(* CODESYS project Avangard(contr1).project
   Title: Avangard(contr1)
   Version: 0.0.0.0
   Author: Administrator

Project tree, tasks and I/O mapping:
  MyController : TM241CE40T/U, Schneider Electric, order no. TM241CE40T/U, version 4.0.6.18
    application Application
      task MAST (cyclic, interval 20 ms, priority 15, watchdog 100 ms x 1) calls MainPrgY, MainLD, MainPrgX
      global variables GVL
    DI : Digital Inputs, Schneider Electric, version 4.0.6.18
        input  idwDI_IDW0 : DWORD  // IDW0
        input  Application.X01_0 : BOOL  // IDW0.I0
        input  Application.X01_1 : BOOL  // IDW0.I1
        input  Application.X01_2 : BOOL  // IDW0.I2
        input  Application.X01_3 : BOOL  // IDW0.I3
        input  Application.X01_4 : BOOL  // IDW0.I4
        input  Application.X01_5 : BOOL  // IDW0.I5
        input  Application.X01_6 : BOOL  // IDW0.I6
        input  Application.X01_7 : BOOL  // IDW0.I7
        input  Application.X01_8 : BOOL  // IDW0.I8
        input  Application.X01_9 : BOOL  // IDW0.I9
        input  Application.X01_10 : BOOL  // IDW0.I10
        input  Application.X01_11 : BOOL  // IDW0.I11
        input  Application.X01_12 : BOOL  // IDW0.I12
        input  Application.X01_13 : BOOL  // IDW0.I13
        input  Application.X01_14 : BOOL  // IDW0.I14
        input  Application.X01_15 : BOOL  // IDW0.I15
        input  Application.X01_16 : BOOL  // IDW0.I16
        input  Application.X01_17 : BOOL  // IDW0.I17
        input  Application.X01_18 : BOOL  // IDW0.I18
        input  Application.X01_19 : BOOL  // IDW0.I19
        input  Application.X01_20 : BOOL  // IDW0.I20
        input  Application.X01_21 : BOOL  // IDW0.I21
        input  Application.X01_22 : BOOL  // IDW0.I22
        input  Application.X01_23 : BOOL  // IDW0.I23
        input  ibDI_IB1 : BYTE  // IB1
    DQ : Digital Outputs, Schneider Electric, version 4.0.6.18
        output Application.Y01_0 : BOOL  // QW0.Q0
        output Application.Y01_1 : BOOL  // QW0.Q1
        output Application.Y01_2 : BOOL  // QW0.Q2
        output Application.Y01_3 : BOOL  // QW0.Q3
        output Application.Y01_4 : BOOL  // QW0.Q4
        output Application.Y01_5 : BOOL  // QW0.Q5
        output Application.Y01_6 : BOOL  // QW0.Q6
        output Application.Y01_7 : BOOL  // QW0.Q7
        output Application.Y01_8 : BOOL  // QW0.Q8
        output Application.Y01_9 : BOOL  // QW0.Q9
        output Application.Y01_10 : BOOL  // QW0.Q10
        output Application.Y01_11 : BOOL  // QW0.Q11
        output Application.Y01_12 : BOOL  // QW0.Q12
        output Application.Y01_13 : BOOL  // QW0.Q13
        output Application.Y01_14 : BOOL  // QW0.Q14
        output Application.Y01_15 : BOOL  // QW0.Q15
        output qbDQ_QB1 : BYTE  // QB1
        unmapped channels: QW0
    Counters : Counters, Schneider Electric, version 4.0.6.18
    Pulse_Generators : Pulse Generators, Schneider Electric, version 4.0.6.18
    Cartridge_1 : Cartridge, Schneider Electric, version 4.0.6.18
    Cartridge_2 : Cartridge, Schneider Electric, version 4.0.6.18
    IO_Bus : IO bus - TM3, Schneider Electric, version 4.0.6.18
      Module_1 : TM3DI32K, Schneider Electric, order no. TM3DI32K, version 1.0.1.3
          input  idwModule_1_ID0 : DWORD  // ID0
          input  Application.X11_0 : BOOL  // ID0.I0
          input  Application.X11_1 : BOOL  // ID0.I1
          input  Application.X11_2 : BOOL  // ID0.I2
          input  Application.X11_3 : BOOL  // ID0.I3
          input  Application.X11_4 : BOOL  // ID0.I4
          input  Application.X11_5 : BOOL  // ID0.I5
          input  Application.X11_6 : BOOL  // ID0.I6
          input  Application.X11_7 : BOOL  // ID0.I7
          input  Application.X11_8 : BOOL  // ID0.I8
          input  Application.X11_9 : BOOL  // ID0.I9
          input  Application.X11_10 : BOOL  // ID0.I10
          input  Application.X11_11 : BOOL  // ID0.I11
          input  Application.X11_12 : BOOL  // ID0.I12
          input  Application.X11_13 : BOOL  // ID0.I13
          input  Application.X11_14 : BOOL  // ID0.I14
          input  Application.X11_15 : BOOL  // ID0.I15
          input  Application.X11_16 : BOOL  // ID0.I16
          input  Application.X11_17 : BOOL  // ID0.I17
          input  Application.X11_18 : BOOL  // ID0.I18
          input  Application.X11_19 : BOOL  // ID0.I19
          input  Application.X11_20 : BOOL  // ID0.I20
          input  Application.X11_21 : BOOL  // ID0.I21
          input  Application.X11_22 : BOOL  // ID0.I22
          input  Application.X11_23 : BOOL  // ID0.I23
          input  Application.X11_24 : BOOL  // ID0.I24
          input  Application.X11_25 : BOOL  // ID0.I25
          input  Application.X11_26 : BOOL  // ID0.I26
          input  Application.X11_27 : BOOL  // ID0.I27
          input  Application.X11_28 : BOOL  // ID0.I28
          input  Application.X11_29 : BOOL  // ID0.I29
          input  Application.X11_30 : BOOL  // ID0.I30
          input  Application.X11_31 : BOOL  // ID0.I31
      Module_2 : TM3DI32K, Schneider Electric, order no. TM3DI32K, version 1.0.1.3
          input  Application.X12_0 : BOOL  // ID0.I0
          input  Application.X12_1 : BOOL  // ID0.I1
          input  Application.X12_2 : BOOL  // ID0.I2
          input  Application.X12_3 : BOOL  // ID0.I3
          input  Application.X12_4 : BOOL  // ID0.I4
          input  Application.X12_5 : BOOL  // ID0.I5
          input  Application.X12_6 : BOOL  // ID0.I6
          input  Application.X12_7 : BOOL  // ID0.I7
          input  Application.X12_8 : BOOL  // ID0.I8
          input  Application.X12_9 : BOOL  // ID0.I9
          input  Application.X12_10 : BOOL  // ID0.I10
          input  Application.X12_11 : BOOL  // ID0.I11
          input  Application.X12_12 : BOOL  // ID0.I12
          input  Application.X12_13 : BOOL  // ID0.I13
          input  Application.X12_14 : BOOL  // ID0.I14
          input  Application.X12_15 : BOOL  // ID0.I15
          input  Application.X12_16 : BOOL  // ID0.I16
          input  Application.X12_17 : BOOL  // ID0.I17
          input  Application.X12_18 : BOOL  // ID0.I18
          input  Application.X12_19 : BOOL  // ID0.I19
          input  Application.X12_20 : BOOL  // ID0.I20
          input  Application.X12_21 : BOOL  // ID0.I21
          input  Application.X12_22 : BOOL  // ID0.I22
          input  Application.X12_23 : BOOL  // ID0.I23
          input  Application.X12_24 : BOOL  // ID0.I24
          input  Application.X12_25 : BOOL  // ID0.I25
          input  Application.X12_26 : BOOL  // ID0.I26
          input  Application.X12_27 : BOOL  // ID0.I27
          input  Application.X12_28 : BOOL  // ID0.I28
          input  Application.X12_29 : BOOL  // ID0.I29
          input  Application.X12_30 : BOOL  // ID0.I30
          input  Application.X12_31 : BOOL  // ID0.I31
          unmapped channels: ID0
      Module_5 : TM3DI32K, Schneider Electric, order no. TM3DI32K, version 1.0.1.3
          input  Application.X15_0 : BOOL  // ID0.I0
          input  Application.X15_1 : BOOL  // ID0.I1
          input  Application.X15_2 : BOOL  // ID0.I2
          input  Application.X15_3 : BOOL  // ID0.I3
          input  Application.X15_4 : BOOL  // ID0.I4
          input  Application.X15_5 : BOOL  // ID0.I5
          input  Application.X15_6 : BOOL  // ID0.I6
          input  Application.X15_7 : BOOL  // ID0.I7
          input  Application.X15_8 : BOOL  // ID0.I8
          input  Application.X15_9 : BOOL  // ID0.I9
          input  Application.X15_10 : BOOL  // ID0.I10
          input  Application.X15_11 : BOOL  // ID0.I11
          input  Application.X15_12 : BOOL  // ID0.I12
          input  Application.X15_13 : BOOL  // ID0.I13
          input  Application.X15_14 : BOOL  // ID0.I14
          input  Application.X15_15 : BOOL  // ID0.I15
          input  Application.X15_16 : BOOL  // ID0.I16
          input  Application.X15_17 : BOOL  // ID0.I17
          input  Application.X15_18 : BOOL  // ID0.I18
          input  Application.X15_19 : BOOL  // ID0.I19
          input  Application.X15_20 : BOOL  // ID0.I20
          input  Application.X15_21 : BOOL  // ID0.I21
          input  Application.X15_22 : BOOL  // ID0.I22
          input  Application.X15_23 : BOOL  // ID0.I23
          input  Application.X15_24 : BOOL  // ID0.I24
          input  Application.X15_25 : BOOL  // ID0.I25
          input  Application.X15_26 : BOOL  // ID0.I26
          input  Application.X15_27 : BOOL  // ID0.I27
          input  Application.X15_28 : BOOL  // ID0.I28
          input  Application.X15_29 : BOOL  // ID0.I29
          input  Application.X15_30 : BOOL  // ID0.I30
          input  Application.X15_31 : BOOL  // ID0.I31
          unmapped channels: ID0
      Module_4 : TM3DI32K, Schneider Electric, order no. TM3DI32K, version 1.0.1.3
          input  Application.X14_0 : BOOL  // ID0.I0
          input  Application.X14_1 : BOOL  // ID0.I1
          input  Application.X14_2 : BOOL  // ID0.I2
          input  Application.X14_3 : BOOL  // ID0.I3
          input  Application.X14_4 : BOOL  // ID0.I4
          input  Application.X14_5 : BOOL  // ID0.I5
          input  Application.X14_6 : BOOL  // ID0.I6
          input  Application.X14_7 : BOOL  // ID0.I7
          input  Application.X14_8 : BOOL  // ID0.I8
          input  Application.X14_9 : BOOL  // ID0.I9
          input  Application.X14_10 : BOOL  // ID0.I10
          input  Application.X14_11 : BOOL  // ID0.I11
          input  Application.X14_12 : BOOL  // ID0.I12
          input  Application.X14_13 : BOOL  // ID0.I13
          input  Application.X14_14 : BOOL  // ID0.I14
          input  Application.X14_15 : BOOL  // ID0.I15
          input  Application.X14_16 : BOOL  // ID0.I16
          input  Application.X14_17 : BOOL  // ID0.I17
          input  Application.X14_18 : BOOL  // ID0.I18
          input  Application.X14_19 : BOOL  // ID0.I19
          input  Application.X14_20 : BOOL  // ID0.I20
          input  Application.X14_21 : BOOL  // ID0.I21
          input  Application.X14_22 : BOOL  // ID0.I22
          input  Application.X14_23 : BOOL  // ID0.I23
          input  Application.X14_24 : BOOL  // ID0.I24
          input  Application.X14_25 : BOOL  // ID0.I25
          input  Application.X14_26 : BOOL  // ID0.I26
          input  Application.X14_27 : BOOL  // ID0.I27
          input  Application.X14_28 : BOOL  // ID0.I28
          input  Application.X14_29 : BOOL  // ID0.I29
          input  Application.X14_30 : BOOL  // ID0.I30
          input  Application.X14_31 : BOOL  // ID0.I31
          unmapped channels: ID0
      Module_3 : TM3DI32K, Schneider Electric, order no. TM3DI32K, version 1.0.1.3
          input  Application.X13_0 : BOOL  // ID0.I0
          input  Application.X13_1 : BOOL  // ID0.I1
          input  Application.X13_2 : BOOL  // ID0.I2
          input  Application.X13_3 : BOOL  // ID0.I3
          input  Application.X13_4 : BOOL  // ID0.I4
          input  Application.X13_5 : BOOL  // ID0.I5
          input  Application.X13_6 : BOOL  // ID0.I6
          input  Application.X13_7 : BOOL  // ID0.I7
          input  Application.X13_8 : BOOL  // ID0.I8
          input  Application.X13_9 : BOOL  // ID0.I9
          input  Application.X13_10 : BOOL  // ID0.I10
          input  Application.X13_11 : BOOL  // ID0.I11
          input  Application.X13_12 : BOOL  // ID0.I12
          input  Application.X13_13 : BOOL  // ID0.I13
          input  Application.X13_14 : BOOL  // ID0.I14
          input  Application.X13_15 : BOOL  // ID0.I15
          input  Application.X13_16 : BOOL  // ID0.I16
          input  Application.X13_17 : BOOL  // ID0.I17
          input  Application.X13_18 : BOOL  // ID0.I18
          input  Application.X13_19 : BOOL  // ID0.I19
          input  Application.X13_20 : BOOL  // ID0.I20
          input  Application.X13_21 : BOOL  // ID0.I21
          input  Application.X13_22 : BOOL  // ID0.I22
          input  Application.X13_23 : BOOL  // ID0.I23
          input  Application.X13_24 : BOOL  // ID0.I24
          input  Application.X13_25 : BOOL  // ID0.I25
          input  Application.X13_26 : BOOL  // ID0.I26
          input  Application.X13_27 : BOOL  // ID0.I27
          input  Application.X13_28 : BOOL  // ID0.I28
          input  Application.X13_29 : BOOL  // ID0.I29
          input  Application.X13_30 : BOOL  // ID0.I30
          input  Application.X13_31 : BOOL  // ID0.I31
          unmapped channels: ID0
      Module_6 : TM3DQ32TK, Schneider Electric, order no. TM3DQ32TK, version 1.0.1.3
          output Application.Y16_0 : BOOL  // QD0.Q0
          output Application.Y16_1 : BOOL  // QD0.Q1
          output Application.Y16_2 : BOOL  // QD0.Q2
          output Application.Y16_3 : BOOL  // QD0.Q3
          output Application.Y16_4 : BOOL  // QD0.Q4
          output Application.Y16_5 : BOOL  // QD0.Q5
          output Application.Y16_6 : BOOL  // QD0.Q6
          output Application.Y16_7 : BOOL  // QD0.Q7
          output Application.Y16_8 : BOOL  // QD0.Q8
          output Application.Y16_9 : BOOL  // QD0.Q9
          output Application.Y16_10 : BOOL  // QD0.Q10
          output Application.Y16_11 : BOOL  // QD0.Q11
          output Application.Y16_12 : BOOL  // QD0.Q12
          output Application.Y16_13 : BOOL  // QD0.Q13
          output Application.Y16_14 : BOOL  // QD0.Q14
          output Application.Y16_15 : BOOL  // QD0.Q15
          output Application.Y16_16 : BOOL  // QD0.Q16
          output Application.Y16_17 : BOOL  // QD0.Q17
          output Application.Y16_18 : BOOL  // QD0.Q18
          output Application.Y16_19 : BOOL  // QD0.Q19
          output Application.Y16_20 : BOOL  // QD0.Q20
          output Application.Y16_21 : BOOL  // QD0.Q21
          output Application.Y16_22 : BOOL  // QD0.Q22
          output Application.Y16_23 : BOOL  // QD0.Q23
          output Application.Y16_24 : BOOL  // QD0.Q24
          output Application.Y16_25 : BOOL  // QD0.Q25
          output Application.Y16_26 : BOOL  // QD0.Q26
          output Application.Y16_27 : BOOL  // QD0.Q27
          output Application.Y16_28 : BOOL  // QD0.Q28
          output Application.Y16_29 : BOOL  // QD0.Q29
          output Application.Y16_30 : BOOL  // QD0.Q30
          output Application.Y16_31 : BOOL  // QD0.Q31
          unmapped channels: QD0
      Module_7 : TM3DQ32TK, Schneider Electric, order no. TM3DQ32TK, version 1.0.1.3
          output Application.Y17_0 : BOOL  // QD0.Q0
          output Application.Y17_1 : BOOL  // QD0.Q1
          output Application.Y17_2 : BOOL  // QD0.Q2
          output Application.Y17_3 : BOOL  // QD0.Q3
          output Application.Y17_4 : BOOL  // QD0.Q4
          output Application.Y17_5 : BOOL  // QD0.Q5
          output Application.Y17_6 : BOOL  // QD0.Q6
          output Application.Y17_7 : BOOL  // QD0.Q7
          output Application.Y17_8 : BOOL  // QD0.Q8
          output Application.Y17_9 : BOOL  // QD0.Q9
          output Application.Y17_10 : BOOL  // QD0.Q10
          output Application.Y17_11 : BOOL  // QD0.Q11
          output Application.Y17_12 : BOOL  // QD0.Q12
          output Application.Y17_13 : BOOL  // QD0.Q13
          output Application.Y17_14 : BOOL  // QD0.Q14
          output Application.Y17_15 : BOOL  // QD0.Q15
          output Application.Y17_16 : BOOL  // QD0.Q16
          output Application.Y17_17 : BOOL  // QD0.Q17
          output Application.Y17_18 : BOOL  // QD0.Q18
          output Application.Y17_19 : BOOL  // QD0.Q19
          output Application.Y17_20 : BOOL  // QD0.Q20
          output Application.Y17_21 : BOOL  // QD0.Q21
          output Application.Y17_22 : BOOL  // QD0.Q22
          output Application.Y17_23 : BOOL  // QD0.Q23
          output Application.Y17_24 : BOOL  // QD0.Q24
          output Application.Y17_25 : BOOL  // QD0.Q25
          output Application.Y17_26 : BOOL  // QD0.Q26
          output Application.Y17_27 : BOOL  // QD0.Q27
          output Application.Y17_28 : BOOL  // QD0.Q28
          output Application.Y17_29 : BOOL  // QD0.Q29
          output Application.Y17_30 : BOOL  // QD0.Q30
          output Application.Y17_31 : BOOL  // QD0.Q31
          unmapped channels: QD0
    COM_Bus : COM bus, Schneider Electric, version 4.0.6.18
    Ethernet_1 : Ethernet Network, Schneider Electric, version 4.0.6.18
        settings: IPAddress = [192, 168, 1, 201]; SubnetMask = [255, 255, 255, 0]; GatewayAddress = [192, 168, 1, 1]; DeviceName = 'TM241CE40T_1'; WebServer = FALSE; FTP Server = FALSE; SoMachine Protocol = TRUE; Modbus Server = TRUE; NetManage Protocol = TRUE; SNMP protocol = FALSE; Enable Routing = FALSE; WebVisu protocol = FALSE; DHCP Server Active = FALSE
    Serial_Line_1 : Serial line, Schneider Electric, version 4.0.6.18
      SoMachine_Network_Manager : SoMachine-Network Manager, Schneider Electric, version 4.0.0.2
    Serial_Line_2 : Serial line, Schneider Electric, version 4.0.6.18
      Modbus_Manager : Modbus Manager, Schneider Electric, version 4.0.0.2
  libraries: Standard, * (System)
  program MainPrgY [ST]
  program MainLD [LD]
  function block DKS [LD]
  program MainPrgX [ST]
*)

// MyController/Application/GVL
VAR_GLOBAL
	XX AT %MW0 : ARRAY[0..11] OF WORD;  //данные с 1го контроллера
	YY AT %MW12 : ARRAY[0..5] OF WORD;  //данные для 1го контроллера на управление

	DKS_Time : WORD := 3;	//время срабатывания ДКС в сек
	
	Nor10200_DKS : BOOL;
	Nor10400_DKS : BOOL;
	Tr10500_DKS : BOOL;
	Tr10600_DKS : BOOL;
	Tr10700_DKS : BOOL;
	Tr20110_DKS : BOOL;
	Nor20300_DKS : BOOL;
	Nor21200_DKS : BOOL;
	Tr21300_DKS : BOOL;
	Tr30400_DKS : BOOL;
	Nor30500_DKS : BOOL;
	Tr30340_DKS : BOOL;
	Tr30700_DKS : BOOL;
	Nor40100_DKS : BOOL;
	
	
	// Контроллер 1
		//Входа
			X01_0 : BOOL;
			X01_1 : BOOL;
			X01_2 : BOOL;
			X01_3 : BOOL;
			X01_4 : BOOL;
			X01_5 : BOOL;
			X01_6 : BOOL;
			X01_7 : BOOL;
			X01_8 : BOOL;
			X01_9 : BOOL;
			X01_10 : BOOL;
			X01_11 : BOOL;
			X01_12 : BOOL;
			X01_13 : BOOL;
			X01_14 : BOOL;
			X01_15 : BOOL;
			X01_16 : BOOL;
			X01_17 : BOOL;
			X01_18 : BOOL;
			X01_19 : BOOL;
			X01_20 : BOOL;
			X01_21 : BOOL;
			X01_22 : BOOL;
			X01_23 : BOOL;
			X01_24 : BOOL;
			X01_25 : BOOL;
			X01_26 : BOOL;
			X01_27 : BOOL;
			X01_28 : BOOL;
			X01_29 : BOOL;
			X01_30 : BOOL;
			X01_31 : BOOL;
		//Выхода
			Y01_0 : BOOL;
			Y01_1 : BOOL;
			Y01_2 : BOOL;
			Y01_3 : BOOL;
			Y01_4 : BOOL;
			Y01_5 : BOOL;
			Y01_6 : BOOL;
			Y01_7 : BOOL;
			Y01_8 : BOOL;
			Y01_9 : BOOL;
			Y01_10 : BOOL;
			Y01_11 : BOOL;
			Y01_12 : BOOL;
			Y01_13 : BOOL;
			Y01_14 : BOOL;
			Y01_15 : BOOL;
			Y01_16 : BOOL;
			Y01_17 : BOOL;
			Y01_18 : BOOL;
			Y01_19 : BOOL;
			Y01_20 : BOOL;
			Y01_21 : BOOL;
			Y01_22 : BOOL;
			Y01_23 : BOOL;
			Y01_24 : BOOL;
			Y01_25 : BOOL;
			Y01_26 : BOOL;
			Y01_27 : BOOL;
			Y01_28 : BOOL;
			Y01_29 : BOOL;
			Y01_30 : BOOL;
			Y01_31 : BOOL;
			
	// Модуль расширения 1 контроллер 1 
		//Входа
			X11_0 : BOOL;
			X11_1 : BOOL;
			X11_2 : BOOL;
			X11_3 : BOOL;
			X11_4 : BOOL;
			X11_5 : BOOL;
			X11_6 : BOOL;
			X11_7 : BOOL;
			X11_8 : BOOL;
			X11_9 : BOOL;
			X11_10 : BOOL;
			X11_11 : BOOL;
			X11_12 : BOOL;
			X11_13 : BOOL;
			X11_14 : BOOL;
			X11_15 : BOOL;
			X11_16 : BOOL;
			X11_17 : BOOL;
			X11_18 : BOOL;
			X11_19 : BOOL;
			X11_20 : BOOL;
			X11_21 : BOOL;
			X11_22 : BOOL;
			X11_23 : BOOL;
			X11_24 : BOOL;
			X11_25 : BOOL;
			X11_26 : BOOL;
			X11_27 : BOOL;
			X11_28 : BOOL;
			X11_29 : BOOL;
			X11_30 : BOOL;
			X11_31 : BOOL;
		//Выхода
			Y11_0 : BOOL;
			Y11_1 : BOOL;
			Y11_2 : BOOL;
			Y11_3 : BOOL;
			Y11_4 : BOOL;
			Y11_5 : BOOL;
			Y11_6 : BOOL;
			Y11_7 : BOOL;
			Y11_8 : BOOL;
			Y11_9 : BOOL;
			Y11_10 : BOOL;
			Y11_11 : BOOL;
			Y11_12 : BOOL;
			Y11_13 : BOOL;
			Y11_14 : BOOL;
			Y11_15 : BOOL;
			Y11_16 : BOOL;
			Y11_17 : BOOL;
			Y11_18 : BOOL;
			Y11_19 : BOOL;
			Y11_20 : BOOL;
			Y11_21 : BOOL;
			Y11_22 : BOOL;
			Y11_23 : BOOL;
			Y11_24 : BOOL;
			Y11_25 : BOOL;
			Y11_26 : BOOL;
			Y11_27 : BOOL;
			Y11_28 : BOOL;
			Y11_29 : BOOL;
			Y11_30 : BOOL;
			Y11_31 : BOOL;
	
	// Модуль расширения 2 контроллер 1
		//Входа
			X12_0 : BOOL;
			X12_1 : BOOL;
			X12_2 : BOOL;
			X12_3 : BOOL;
			X12_4 : BOOL;
			X12_5 : BOOL;
			X12_6 : BOOL;
			X12_7 : BOOL;
			X12_8 : BOOL;
			X12_9 : BOOL;
			X12_10 : BOOL;
			X12_11 : BOOL;
			X12_12 : BOOL;
			X12_13 : BOOL;
			X12_14 : BOOL;
			X12_15 : BOOL;
			X12_16 : BOOL;
			X12_17 : BOOL;
			X12_18 : BOOL;
			X12_19 : BOOL;
			X12_20 : BOOL;
			X12_21 : BOOL;
			X12_22 : BOOL;
			X12_23 : BOOL;
			X12_24 : BOOL;
			X12_25 : BOOL;
			X12_26 : BOOL;
			X12_27 : BOOL;
			X12_28 : BOOL;
			X12_29 : BOOL;
			X12_30 : BOOL;
			X12_31 : BOOL;
		//Выхода
			Y12_0 : BOOL;
			Y12_1 : BOOL;
			Y12_2 : BOOL;
			Y12_3 : BOOL;
			Y12_4 : BOOL;
			Y12_5 : BOOL;
			Y12_6 : BOOL;
			Y12_7 : BOOL;
			Y12_8 : BOOL;
			Y12_9 : BOOL;
			Y12_10 : BOOL;
			Y12_11 : BOOL;
			Y12_12 : BOOL;
			Y12_13 : BOOL;
			Y12_14 : BOOL;
			Y12_15 : BOOL;
			Y12_16 : BOOL;
			Y12_17 : BOOL;
			Y12_18 : BOOL;
			Y12_19 : BOOL;
			Y12_20 : BOOL;
			Y12_21 : BOOL;
			Y12_22 : BOOL;
			Y12_23 : BOOL;
			Y12_24 : BOOL;
			Y12_25 : BOOL;
			Y12_26 : BOOL;
			Y12_27 : BOOL;
			Y12_28 : BOOL;
			Y12_29 : BOOL;
			Y12_30 : BOOL;
			Y12_31 : BOOL;
			
	// Модуль расширения 3 контроллер 1
		//Входа
			X13_0 : BOOL;
			X13_1 : BOOL;
			X13_2 : BOOL;
			X13_3 : BOOL;
			X13_4 : BOOL;
			X13_5 : BOOL;
			X13_6 : BOOL;
			X13_7 : BOOL;
			X13_8 : BOOL;
			X13_9 : BOOL;
			X13_10 : BOOL;
			X13_11 : BOOL;
			X13_12 : BOOL;
			X13_13 : BOOL;
			X13_14 : BOOL;
			X13_15 : BOOL;
			X13_16 : BOOL;
			X13_17 : BOOL;
			X13_18 : BOOL;
			X13_19 : BOOL;
			X13_20 : BOOL;
			X13_21 : BOOL;
			X13_22 : BOOL;
			X13_23 : BOOL;
			X13_24 : BOOL;
			X13_25 : BOOL;
			X13_26 : BOOL;
			X13_27 : BOOL;
			X13_28 : BOOL;
			X13_29 : BOOL;
			X13_30 : BOOL;
			X13_31 : BOOL;
		//Выхода
			Y13_0 : BOOL;
			Y13_1 : BOOL;
			Y13_2 : BOOL;
			Y13_3 : BOOL;
			Y13_4 : BOOL;
			Y13_5 : BOOL;
			Y13_6 : BOOL;
			Y13_7 : BOOL;
			Y13_8 : BOOL;
			Y13_9 : BOOL;
			Y13_10 : BOOL;
			Y13_11 : BOOL;
			Y13_12 : BOOL;
			Y13_13 : BOOL;
			Y13_14 : BOOL;
			Y13_15 : BOOL;
			Y13_16 : BOOL;
			Y13_17 : BOOL;
			Y13_18 : BOOL;
			Y13_19 : BOOL;
			Y13_20 : BOOL;
			Y13_21 : BOOL;
			Y13_22 : BOOL;
			Y13_23 : BOOL;
			Y13_24 : BOOL;
			Y13_25 : BOOL;
			Y13_26 : BOOL;
			Y13_27 : BOOL;
			Y13_28 : BOOL;
			Y13_29 : BOOL;
			Y13_30 : BOOL;
			Y13_31 : BOOL;			

	// Модуль расширения 4 контроллер 1
		//Входа
			X14_0 : BOOL;
			X14_1 : BOOL;
			X14_2 : BOOL;
			X14_3 : BOOL;
			X14_4 : BOOL;
			X14_5 : BOOL;
			X14_6 : BOOL;
			X14_7 : BOOL;
			X14_8 : BOOL;
			X14_9 : BOOL;
			X14_10 : BOOL;
			X14_11 : BOOL;
			X14_12 : BOOL;
			X14_13 : BOOL;
			X14_14 : BOOL;
			X14_15 : BOOL;
			X14_16 : BOOL;
			X14_17 : BOOL;
			X14_18 : BOOL;
			X14_19 : BOOL;
			X14_20 : BOOL;
			X14_21 : BOOL;
			X14_22 : BOOL;
			X14_23 : BOOL;
			X14_24 : BOOL;
			X14_25 : BOOL;
			X14_26 : BOOL;
			X14_27 : BOOL;
			X14_28 : BOOL;
			X14_29 : BOOL;
			X14_30 : BOOL;
			X14_31 : BOOL;
		//Выхода
			Y14_0 : BOOL;
			Y14_1 : BOOL;
			Y14_2 : BOOL;
			Y14_3 : BOOL;
			Y14_4 : BOOL;
			Y14_5 : BOOL;
			Y14_6 : BOOL;
			Y14_7 : BOOL;
			Y14_8 : BOOL;
			Y14_9 : BOOL;
			Y14_10 : BOOL;
			Y14_11 : BOOL;
			Y14_12 : BOOL;
			Y14_13 : BOOL;
			Y14_14 : BOOL;
			Y14_15 : BOOL;
			Y14_16 : BOOL;
			Y14_17 : BOOL;
			Y14_18 : BOOL;
			Y14_19 : BOOL;
			Y14_20 : BOOL;
			Y14_21 : BOOL;
			Y14_22 : BOOL;
			Y14_23 : BOOL;
			Y14_24 : BOOL;
			Y14_25 : BOOL;
			Y14_26 : BOOL;
			Y14_27 : BOOL;
			Y14_28 : BOOL;
			Y14_29 : BOOL;
			Y14_30 : BOOL;
			Y14_31 : BOOL;
	// Модуль расширения 5 контроллер 1
		//Входа
			X15_0 : BOOL;
			X15_1 : BOOL;
			X15_2 : BOOL;
			X15_3 : BOOL;
			X15_4 : BOOL;
			X15_5 : BOOL;
			X15_6 : BOOL;
			X15_7 : BOOL;
			X15_8 : BOOL;
			X15_9 : BOOL;
			X15_10 : BOOL;
			X15_11 : BOOL;
			X15_12 : BOOL;
			X15_13 : BOOL;
			X15_14 : BOOL;
			X15_15 : BOOL;
			X15_16 : BOOL;
			X15_17 : BOOL;
			X15_18 : BOOL;
			X15_19 : BOOL;
			X15_20 : BOOL;
			X15_21 : BOOL;
			X15_22 : BOOL;
			X15_23 : BOOL;
			X15_24 : BOOL;
			X15_25 : BOOL;
			X15_26 : BOOL;
			X15_27 : BOOL;
			X15_28 : BOOL;
			X15_29 : BOOL;
			X15_30 : BOOL;
			X15_31 : BOOL;
		//Выхода
			Y15_0 : BOOL;
			Y15_1 : BOOL;
			Y15_2 : BOOL;
			Y15_3 : BOOL;
			Y15_4 : BOOL;
			Y15_5 : BOOL;
			Y15_6 : BOOL;
			Y15_7 : BOOL;
			Y15_8 : BOOL;
			Y15_9 : BOOL;
			Y15_10 : BOOL;
			Y15_11 : BOOL;
			Y15_12 : BOOL;
			Y15_13 : BOOL;
			Y15_14 : BOOL;
			Y15_15 : BOOL;
			Y15_16 : BOOL;
			Y15_17 : BOOL;
			Y15_18 : BOOL;
			Y15_19 : BOOL;
			Y15_20 : BOOL;
			Y15_21 : BOOL;
			Y15_22 : BOOL;
			Y15_23 : BOOL;
			Y15_24 : BOOL;
			Y15_25 : BOOL;
			Y15_26 : BOOL;
			Y15_27 : BOOL;
			Y15_28 : BOOL;
			Y15_29 : BOOL;
			Y15_30 : BOOL;
			Y15_31 : BOOL;
	// Модуль расширения 6 контроллер 1
		//Входа
			X16_0 : BOOL;
			X16_1 : BOOL;
			X16_2 : BOOL;
			X16_3 : BOOL;
			X16_4 : BOOL;
			X16_5 : BOOL;
			X16_6 : BOOL;
			X16_7 : BOOL;
			X16_8 : BOOL;
			X16_9 : BOOL;
			X16_10 : BOOL;
			X16_11 : BOOL;
			X16_12 : BOOL;
			X16_13 : BOOL;
			X16_14 : BOOL;
			X16_15 : BOOL;
			X16_16 : BOOL;
			X16_17 : BOOL;
			X16_18 : BOOL;
			X16_19 : BOOL;
			X16_20 : BOOL;
			X16_21 : BOOL;
			X16_22 : BOOL;
			X16_23 : BOOL;
			X16_24 : BOOL;
			X16_25 : BOOL;
			X16_26 : BOOL;
			X16_27 : BOOL;
			X16_28 : BOOL;
			X16_29 : BOOL;
			X16_30 : BOOL;
			X16_31 : BOOL;
		//Выхода
			Y16_0 : BOOL;
			Y16_1 : BOOL;
			Y16_2 : BOOL;
			Y16_3 : BOOL;
			Y16_4 : BOOL;
			Y16_5 : BOOL;
			Y16_6 : BOOL;
			Y16_7 : BOOL;
			Y16_8 : BOOL;
			Y16_9 : BOOL;
			Y16_10 : BOOL;
			Y16_11 : BOOL;
			Y16_12 : BOOL;
			Y16_13 : BOOL;
			Y16_14 : BOOL;
			Y16_15 : BOOL;
			Y16_16 : BOOL;
			Y16_17 : BOOL;
			Y16_18 : BOOL;
			Y16_19 : BOOL;
			Y16_20 : BOOL;
			Y16_21 : BOOL;
			Y16_22 : BOOL;
			Y16_23 : BOOL;
			Y16_24 : BOOL;
			Y16_25 : BOOL;
			Y16_26 : BOOL;
			Y16_27 : BOOL;
			Y16_28 : BOOL;
			Y16_29 : BOOL;
			Y16_30 : BOOL;
			Y16_31 : BOOL;

	// Модуль расширения 7 контроллер 1
		//Входа
			X17_0 : BOOL;
			X17_1 : BOOL;
			X17_2 : BOOL;
			X17_3 : BOOL;
			X17_4 : BOOL;
			X17_5 : BOOL;
			X17_6 : BOOL;
			X17_7 : BOOL;
			X17_8 : BOOL;
			X17_9 : BOOL;
			X17_10 : BOOL;
			X17_11 : BOOL;
			X17_12 : BOOL;
			X17_13 : BOOL;
			X17_14 : BOOL;
			X17_15 : BOOL;
			X17_16 : BOOL;
			X17_17 : BOOL;
			X17_18 : BOOL;
			X17_19 : BOOL;
			X17_20 : BOOL;
			X17_21 : BOOL;
			X17_22 : BOOL;
			X17_23 : BOOL;
			X17_24 : BOOL;
			X17_25 : BOOL;
			X17_26 : BOOL;
			X17_27 : BOOL;
			X17_28 : BOOL;
			X17_29 : BOOL;
			X17_30 : BOOL;
			X17_31 : BOOL;
		//Выхода
			Y17_0 : BOOL;
			Y17_1 : BOOL;
			Y17_2 : BOOL;
			Y17_3 : BOOL;
			Y17_4 : BOOL;
			Y17_5 : BOOL;
			Y17_6 : BOOL;
			Y17_7 : BOOL;
			Y17_8 : BOOL;
			Y17_9 : BOOL;
			Y17_10 : BOOL;
			Y17_11 : BOOL;
			Y17_12 : BOOL;
			Y17_13 : BOOL;
			Y17_14 : BOOL;
			Y17_15 : BOOL;
			Y17_16 : BOOL;
			Y17_17 : BOOL;
			Y17_18 : BOOL;
			Y17_19 : BOOL;
			Y17_20 : BOOL;
			Y17_21 : BOOL;
			Y17_22 : BOOL;
			Y17_23 : BOOL;
			Y17_24 : BOOL;
			Y17_25 : BOOL;
			Y17_26 : BOOL;
			Y17_27 : BOOL;
			Y17_28 : BOOL;
			Y17_29 : BOOL;
			Y17_30 : BOOL;
			Y17_31 : BOOL;

END_VAR

// MainPrgY
PROGRAM MainPrgY
VAR
END_VAR

	//выходы
		Y01_0 := YY[0].0;		
		Y01_1 := YY[0].1;
		Y01_2 := YY[0].2;
		Y01_3 := YY[0].3;
		Y01_4 := YY[0].4;
		Y01_5 := YY[0].5;
		Y01_6 := YY[0].6;
		Y01_7 := YY[0].7;
		Y01_8 := YY[0].8;
		Y01_9 := YY[0].9;
		Y01_10 := YY[0].10;
		Y01_11 := YY[0].11;
		Y01_12 := YY[0].12;
		Y01_13 := YY[0].13;
		Y01_14 := YY[0].14;
		Y01_15 := YY[0].15;
		Y01_16 := YY[1].0;
		Y01_17 := YY[1].1;
		Y01_18 := YY[1].2;
		Y01_19 := YY[1].3;
		Y01_20 := YY[1].4;
		Y01_21 := YY[1].5;
		Y01_22 := YY[1].6;
		Y01_23 := YY[1].7;
		Y01_24 := YY[1].8;
		Y01_25 := YY[1].9;
		Y01_26 := YY[1].10;
		Y01_27 := YY[1].11;
		Y01_28 := YY[1].12;
		Y01_29 := YY[1].13;
		Y01_30 := YY[1].14;
		Y01_31 := YY[1].15;
		
		Y16_0 := YY[2].0;		
		Y16_1 := YY[2].1;
		Y16_2 := YY[2].2;
		Y16_3 := YY[2].3;
		Y16_4 := YY[2].4;
		Y16_5 := YY[2].5;
		Y16_6 := YY[2].6;
		Y16_7 := YY[2].7;
		Y16_8 := YY[2].8;
		Y16_9 := YY[2].9;
		Y16_10 := YY[2].10;
		Y16_11 := YY[2].11;
		Y16_12 := YY[2].12;
		Y16_13 := YY[2].13;
		Y16_14 := YY[2].14;
		Y16_15 := YY[2].15;
		Y16_16 := YY[3].0;
		Y16_17 := YY[3].1;
		Y16_18 := YY[3].2;
		Y16_19 := YY[3].3;
		Y16_20 := YY[3].4;
		Y16_21 := YY[3].5;
		Y16_22 := YY[3].6;
		Y16_23 := YY[3].7;
		Y16_24 := YY[3].8;
		Y16_25 := YY[3].9;
		Y16_26 := YY[3].10;
		Y16_27 := YY[3].11;
		Y16_28 := YY[3].12;
		Y16_29 := YY[3].13;
		Y16_30 := YY[3].14;
		Y16_31 := YY[3].15;
		
		Y17_0 := YY[4].0;		
		Y17_1 := YY[4].1;
		Y17_2 := YY[4].2;
		Y17_3 := YY[4].3;
		Y17_4 := YY[4].4;
		Y17_5 := YY[4].5;
		Y17_6 := YY[4].6;
		Y17_7 := YY[4].7;
		Y17_8 := YY[4].8;
		Y17_9 := YY[4].9;
		Y17_10 := YY[4].10;
		Y17_11 := YY[4].11;
		Y17_12 := YY[4].12;
		Y17_13 := YY[4].13;
		Y17_14 := YY[4].14;
		Y17_15 := YY[4].15;
		Y17_16 := YY[5].0;
		Y17_17 := YY[5].1;
		Y17_18 := YY[5].2;
		Y17_19 := YY[5].3;
		Y17_20 := YY[5].4;
		Y17_21 := YY[5].5;
		Y17_22 := YY[5].6;
		Y17_23 := YY[5].7;
		Y17_24 := YY[5].8;
		Y17_25 := YY[5].9;
		Y17_26 := YY[5].10;
		Y17_27 := YY[5].11;
		Y17_28 := YY[5].12;
		Y17_29 := YY[5].13;
		Y17_30 := YY[5].14;
		Y17_31 := YY[5].15;

END_PROGRAM

// MainLD
PROGRAM MainLD
VAR
	DKS_Nor10200: DKS;
	DKS_Nor10400: DKS;
	DKS_Tr10500: DKS;
	DKS_Tr10600: DKS;
	DKS_Tr10700: DKS;
	DKS_Tr20110: DKS;
	DKS_Nor20300: DKS;
	DKS_Nor21200: DKS;
	DKS_Tr21300: DKS;
	DKS_Tr30400: DKS;
	DKS_Nor30500: DKS;
	DKS_Tr30340: DKS;
	DKS_Tr30700: DKS;
	DKS_Nor40100: DKS;
END_VAR

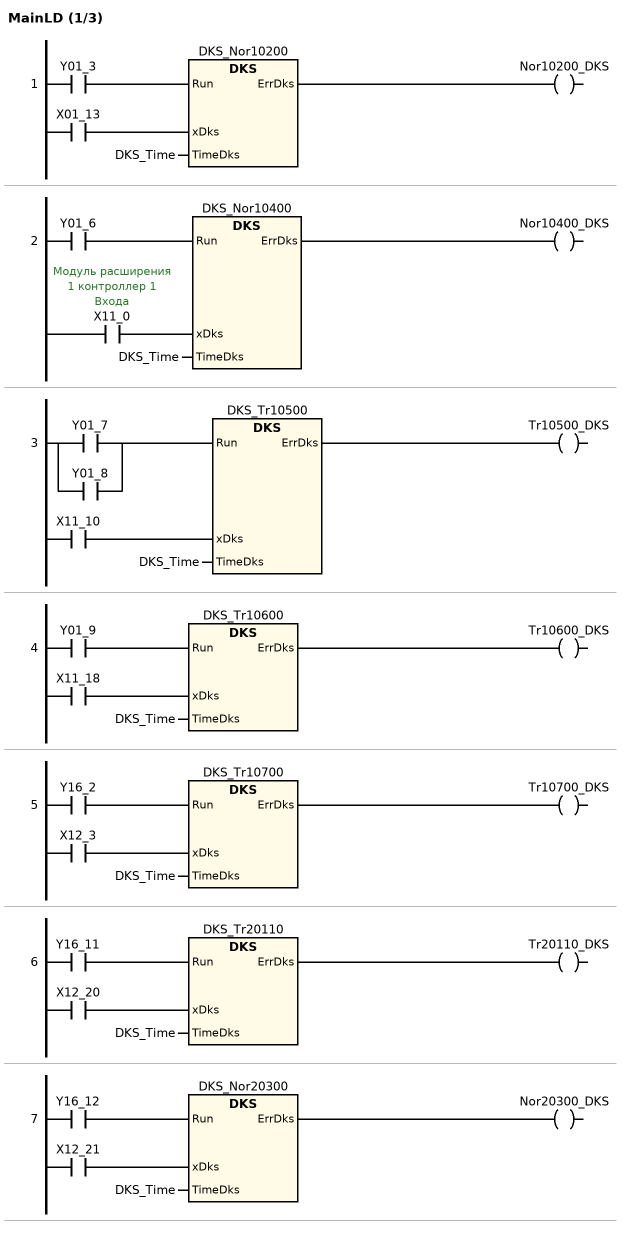
// NETWORK 1
//   DKS_Time: время срабатывания ДКС в сек
DKS_Nor10200(Run := Y01_3, xDks := X01_13, TimeDks := DKS_Time); // DKS
Nor10200_DKS := DKS_Nor10200.ErrDks;

// NETWORK 2
//   X11_0: Модуль расширения 1 контроллер 1 Входа
//   DKS_Time: время срабатывания ДКС в сек
DKS_Nor10400(Run := Y01_6, xDks := X11_0, TimeDks := DKS_Time); // DKS
Nor10400_DKS := DKS_Nor10400.ErrDks;

// NETWORK 3
//   DKS_Time: время срабатывания ДКС в сек
DKS_Tr10500(Run := Y01_7 OR Y01_8, xDks := X11_10, TimeDks := DKS_Time); // DKS
Tr10500_DKS := DKS_Tr10500.ErrDks;

// NETWORK 4
//   DKS_Time: время срабатывания ДКС в сек
DKS_Tr10600(Run := Y01_9, xDks := X11_18, TimeDks := DKS_Time); // DKS
Tr10600_DKS := DKS_Tr10600.ErrDks;

// NETWORK 5
//   DKS_Time: время срабатывания ДКС в сек
DKS_Tr10700(Run := Y16_2, xDks := X12_3, TimeDks := DKS_Time); // DKS
Tr10700_DKS := DKS_Tr10700.ErrDks;

// NETWORK 6
//   DKS_Time: время срабатывания ДКС в сек
DKS_Tr20110(Run := Y16_11, xDks := X12_20, TimeDks := DKS_Time); // DKS
Tr20110_DKS := DKS_Tr20110.ErrDks;

// NETWORK 7
//   DKS_Time: время срабатывания ДКС в сек
DKS_Nor20300(Run := Y16_12, xDks := X12_21, TimeDks := DKS_Time); // DKS
Nor20300_DKS := DKS_Nor20300.ErrDks;

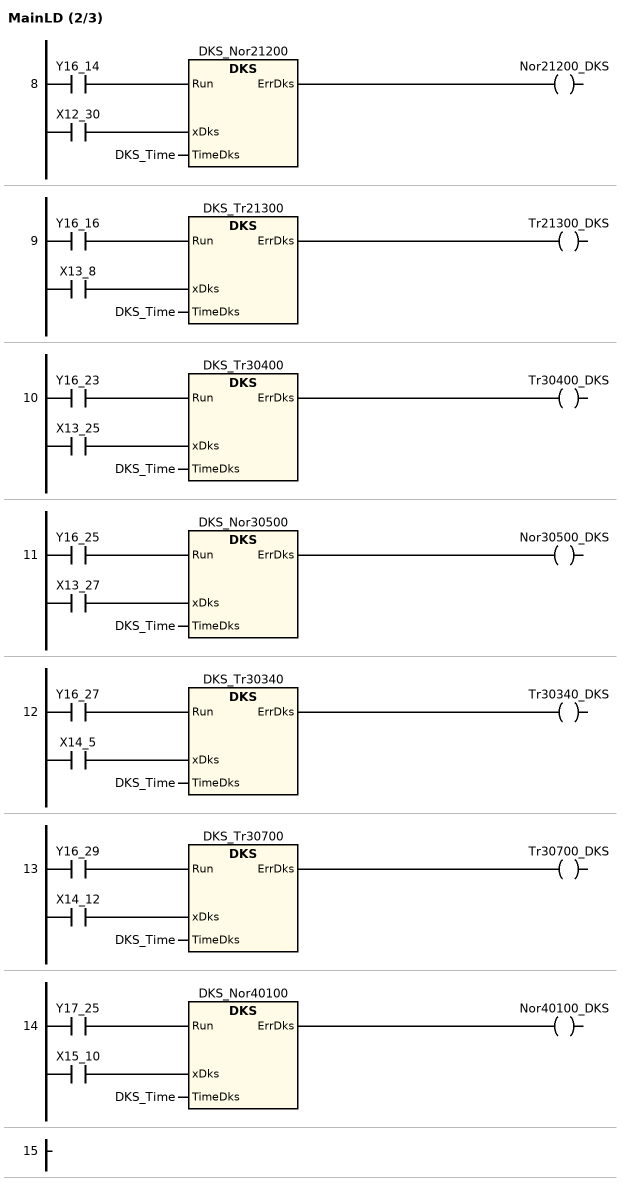
// NETWORK 8
//   DKS_Time: время срабатывания ДКС в сек
DKS_Nor21200(Run := Y16_14, xDks := X12_30, TimeDks := DKS_Time); // DKS
Nor21200_DKS := DKS_Nor21200.ErrDks;

// NETWORK 9
//   DKS_Time: время срабатывания ДКС в сек
DKS_Tr21300(Run := Y16_16, xDks := X13_8, TimeDks := DKS_Time); // DKS
Tr21300_DKS := DKS_Tr21300.ErrDks;

// NETWORK 10
//   DKS_Time: время срабатывания ДКС в сек
DKS_Tr30400(Run := Y16_23, xDks := X13_25, TimeDks := DKS_Time); // DKS
Tr30400_DKS := DKS_Tr30400.ErrDks;

// NETWORK 11
//   DKS_Time: время срабатывания ДКС в сек
DKS_Nor30500(Run := Y16_25, xDks := X13_27, TimeDks := DKS_Time); // DKS
Nor30500_DKS := DKS_Nor30500.ErrDks;

// NETWORK 12
//   DKS_Time: время срабатывания ДКС в сек
DKS_Tr30340(Run := Y16_27, xDks := X14_5, TimeDks := DKS_Time); // DKS
Tr30340_DKS := DKS_Tr30340.ErrDks;

// NETWORK 13
//   DKS_Time: время срабатывания ДКС в сек
DKS_Tr30700(Run := Y16_29, xDks := X14_12, TimeDks := DKS_Time); // DKS
Tr30700_DKS := DKS_Tr30700.ErrDks;

// NETWORK 14
//   DKS_Time: время срабатывания ДКС в сек
DKS_Nor40100(Run := Y17_25, xDks := X15_10, TimeDks := DKS_Time); // DKS
Nor40100_DKS := DKS_Nor40100.ErrDks;

// NETWORK 15

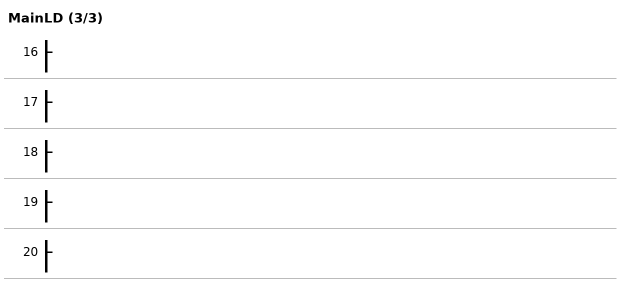
// NETWORK 16

// NETWORK 17

// NETWORK 18

// NETWORK 19

// NETWORK 20

END_PROGRAM

// DKS
FUNCTION_BLOCK DKS
VAR_INPUT
	Run : BOOL;
	xDks : BOOL;
	TimeDks : WORD;
END_VAR

VAR_OUTPUT
	ErrDks : BOOL;
END_VAR
VAR
	TON_DKS_ON: TON;
	TON_DKS_OFF: TON;
END_VAR

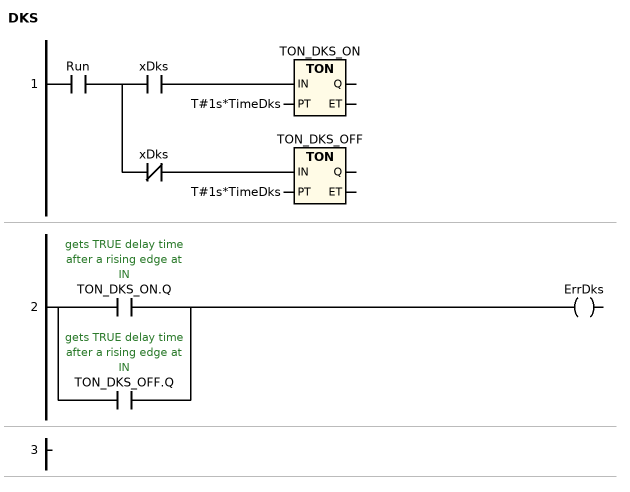
// NETWORK 1
TON_DKS_ON(IN := Run AND xDks, PT := T#1s*TimeDks); // TON
TON_DKS_OFF(IN := Run AND NOT xDks, PT := T#1s*TimeDks); // TON

// NETWORK 2
//   TON_DKS_ON.Q: gets TRUE delay time after a rising edge at IN
//   TON_DKS_OFF.Q: gets TRUE delay time after a rising edge at IN
ErrDks := TON_DKS_ON.Q OR TON_DKS_OFF.Q;

// NETWORK 3

END_FUNCTION_BLOCK

// MainPrgX
PROGRAM MainPrgX
VAR
END_VAR

		XX[0].0 := X01_0;
		XX[0].1 := X01_1;
		XX[0].2 := X01_2;
		XX[0].3 := X01_3;
		XX[0].4 := X01_4;
		XX[0].5 := X01_5;
		XX[0].6 := X01_6;
		XX[0].7 := X01_7;
		XX[0].8 := X01_8;
		XX[0].9 := X01_9;
		XX[0].10 := X01_10;
		XX[0].11 := X01_11;
		XX[0].12 := X01_12;
		XX[0].13 := Nor10200_DKS;	//X01_13;
		XX[0].14 := X01_14;
		XX[0].15 := X01_15;
		XX[1].0 := X01_16;
		XX[1].1 := X01_17;
		XX[1].2 := X01_18;
		XX[1].3 := X01_19;
		XX[1].4 := X01_20;
		XX[1].5 := X01_21;
		XX[1].6 := X01_22;
		XX[1].7 := X01_23;
		XX[1].8 := X01_24;
		XX[1].9 := X01_25;
		XX[1].10 := X01_26;
		XX[1].11 := X01_27;
		XX[1].12 := X01_28;
		XX[1].13 := X01_29;
		XX[1].14 := X01_30;
		XX[1].15 := X01_31;
		
		XX[2].0 := Nor10400_DKS;	//X11_0;
		XX[2].1 := X11_1;
		XX[2].2 := X11_2;
		XX[2].3 := X11_3;
		XX[2].4 := X11_4;
		XX[2].5 := X11_5;
		XX[2].6 := X11_6;
		XX[2].7 := X11_7;
		XX[2].8 := X11_8;
		XX[2].9 := X11_9;
		XX[2].10 := Tr10500_DKS;	//X11_10;
		XX[2].11 := X11_11;
		XX[2].12 := X11_12;
		XX[2].13 := X11_13;
		XX[2].14 := X11_14;
		XX[2].15 := X11_15;
		XX[3].0 := X11_16;
		XX[3].1 := X11_17;
		XX[3].2 := Tr10600_DKS;		//X11_18;
		XX[3].3 := X11_19;
		XX[3].4 := X11_20;
		XX[3].5 := X11_21;
		XX[3].6 := X11_22;
		XX[3].7 := X11_23;
		XX[3].8 := X11_24;
		XX[3].9 := X11_25;
		XX[3].10 := X11_26;
		XX[3].11 := X11_27;
		XX[3].12 := X11_28;
		XX[3].13 := X11_29;
		XX[3].14 := X11_30;
		XX[3].15 := X11_31;
		
		XX[4].0 := X12_0;
		XX[4].1 := X12_1;
		XX[4].2 := X12_2;
		XX[4].3 := Tr10700_DKS;		//X12_3;
		XX[4].4 := X12_4;
		XX[4].5 := X12_5;
		XX[4].6 := X12_6;
		XX[4].7 := X12_7;
		XX[4].8 := X12_8;
		XX[4].9 := X12_9;
		XX[4].10 := X12_10;
		XX[4].11 := X12_11;
		XX[4].12 := X12_12;
		XX[4].13 := X12_13;
		XX[4].14 := X12_14;
		XX[4].15 := X12_15;
		XX[5].0 := X12_16;
		XX[5].1 := X12_17;
		XX[5].2 := X12_18;
		XX[5].3 := X12_19;
		XX[5].4 := Tr20110_DKS;		//X12_20;
		XX[5].5 := Nor20300_DKS;	//X12_21;
		XX[5].6 := X12_22;
		XX[5].7 := X12_23;
		XX[5].8 := X12_24;
		XX[5].9 := X12_25;
		XX[5].10 := X12_26;
		XX[5].11 := X12_27;
		XX[5].12 := X12_28;
		XX[5].13 := X12_29;
		XX[5].14 := Nor21200_DKS;	//X12_30;
		XX[5].15 := X12_31;
		
		XX[6].0 := X13_0;
		XX[6].1 := X13_1;
		XX[6].2 := X13_2;
		XX[6].3 := X13_3;
		XX[6].4 := X13_4;
		XX[6].5 := X13_5;
		XX[6].6 := X13_6;
		XX[6].7 := X13_7;
		XX[6].8 := Tr21300_DKS;		//X13_8;
		XX[6].9 := X13_9;
		XX[6].10 := X13_10;
		XX[6].11 := X13_11;
		XX[6].12 := X13_12;
		XX[6].13 := X13_13;
		XX[6].14 := X13_14;
		XX[6].15 := X13_15;
		XX[7].0 := X13_16;
		XX[7].1 := X13_17;
		XX[7].2 := X13_18;
		XX[7].3 := X13_19;
		XX[7].4 := X13_20;
		XX[7].5 := X13_21;
		XX[7].6 := X13_22;
		XX[7].7 := X13_23;
		XX[7].8 := X13_24;
		XX[7].9 := Tr30400_DKS;		//X13_25;
		XX[7].10 := X13_26;
		XX[7].11 := Nor30500_DKS;	//X13_27;
		XX[7].12 := X13_28;
		XX[7].13 := X13_29;
		XX[7].14 := X13_30;
		XX[7].15 := X13_31;
		
		XX[8].0 := X14_0;
		XX[8].1 := X14_1;
		XX[8].2 := X14_2;
		XX[8].3 := X14_3;
		XX[8].4 := X14_4;
		XX[8].5 := Tr30340_DKS;		//X14_5;
		XX[8].6 := X14_6;
		XX[8].7 := X14_7;
		XX[8].8 := X14_8;
		XX[8].9 := X14_9;
		XX[8].10 := X14_10;
		XX[8].11 := X14_11;
		XX[8].12 := Tr30700_DKS;	//X14_12;
		XX[8].13 := X14_13;
		XX[8].14 := X14_14;
		XX[8].15 := X14_15;
		XX[9].0 := X14_16;
		XX[9].1 := X14_17;
		XX[9].2 := X14_18;
		XX[9].3 := X14_19;
		XX[9].4 := X14_20;
		XX[9].5 := X14_21;
		XX[9].6 := X14_22;
		XX[9].7 := X14_23;
		XX[9].8 := X14_24;
		XX[9].9 := X14_25;
		XX[9].10 := X14_26;
		XX[9].11 := X14_27;
		XX[9].12 := X14_28;
		XX[9].13 := X14_29;
		XX[9].14 := X14_30;
		XX[9].15 := X14_31;
		
		XX[10].0 := X15_0;
		XX[10].1 := X15_1;
		XX[10].2 := X15_2;
		XX[10].3 := X15_3;
		XX[10].4 := X15_4;
		XX[10].5 := X15_5;
		XX[10].6 := X15_6;
		XX[10].7 := X15_7;
		XX[10].8 := X15_8;
		XX[10].9 := X15_9;
		XX[10].10 := Nor40100_DKS;	//X15_10;
		XX[10].11 := X15_11;
		XX[10].12 := X15_12;
		XX[10].13 := X15_13;
		XX[10].14 := X15_14;
		XX[10].15 := X15_15;
		XX[11].0 := X15_16;
		XX[11].1 := X15_17;
		XX[11].2 := X15_18;
		XX[11].3 := X15_19;
		XX[11].4 := X15_20;
		XX[11].5 := X15_21;
		XX[11].6 := X15_22;
		XX[11].7 := X15_23;
		XX[11].8 := X15_24;
		XX[11].9 := X15_25;
		XX[11].10 := X15_26;
		XX[11].11 := X15_27;
		XX[11].12 := X15_28;
		XX[11].13 := X15_29;
		XX[11].14 := X15_30;
		XX[11].15 := X15_31;

END_PROGRAM
